PROGRAM MAIN
VAR
END_VAR

END_PROGRAM

(* stored: Version 1.1.0.1
   POU MAIN: Id {5900ec57-aa3d-4b6a-bde0-4d1931ef6dd0} *)
